// TIA Portal V19 export
DATA_BLOCK "PUMP SELECTION"   // DB36
{ S7_Optimized_Access := 'FALSE' }
   VAR RETAIN
      "P-202 A RO 1 FEED PUMP" : Bool;
      "P-202 B RO 1 FEED PUMP" : Bool;
      "P-202 C RO 1 FEED PUMP" : Bool;
      "P-301 RO 1 HPP PUMP A" : Bool;
      "P-301 RO 1 HPP PUMP B" : Bool;
      "P-401 A RO 2 FEED PUMP" : Bool;
      "P-401 B RO 2 FEED PUMP" : Bool;
      "P-401 C RO 2 FEED PUMP" : Bool;
      "P-402 RO 2 HPP A" : Bool;
      "P-402 RO 2 HPP B" : Bool;
      "P-501 A EDI FEED PUMP" : Bool;
      "P-501 B EDI FEED PUMP" : Bool;
      "P-501 C EDI FEED PUMP" : Bool;
      "EDI-501" : Bool;
      "EDI-502" : Bool;
   END_VAR
BEGIN
END_DATA_BLOCK
